{attribute 'qualified_only' := ''}
VAR_GLOBAL CONSTANT
(*******************************************************************)
(* Globale KONSTANTEN *)
(*******************************************************************)
END_VAR

(* stored: Version 1.1.0.1, ProductVersion 3.1.4024.6
   GVL CONST: Id {43949239-8437-4dc7-99ab-7b2f7f8336e3} *)
